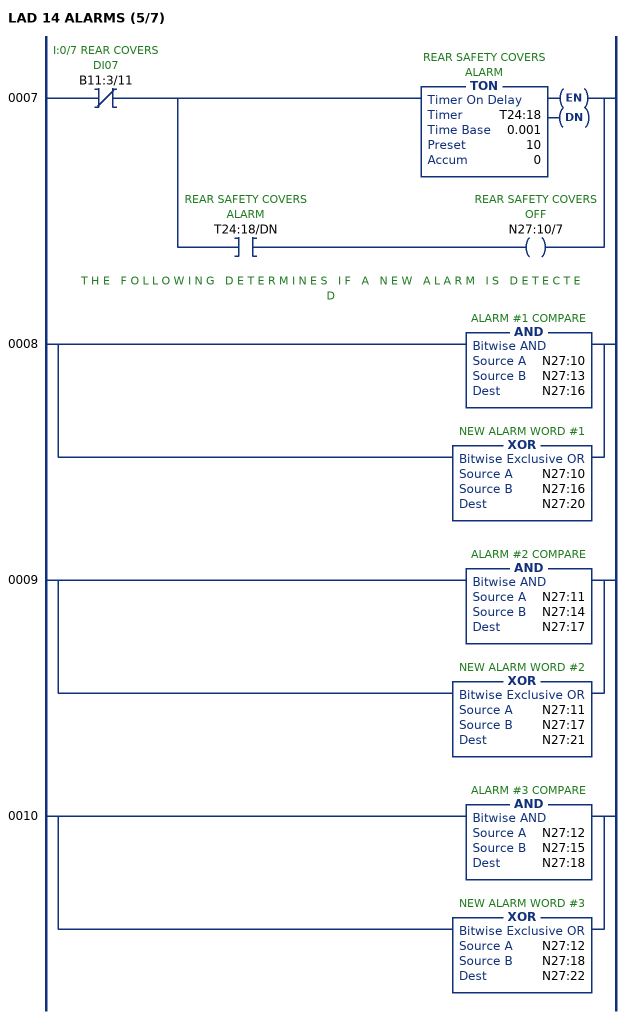
% Rung: 7 %
SOR XIO B11:3/11 BST TON T24:18 0.001 10 0 NXB XIC T24:18/DN OTE N27:10/7 BND EOR
%   B11:3/11  DI07  "I:0/7 REAR COVERS" %
%   T24:18  "REAR SAFETY COVERS ALARM" %
%   N27:10/7  "REAR SAFETY COVERS OFF" %
% Rung: 8 %
%        T H E   F O L L O W I N G   D E T E R M I N E S   I F   A   N E W   A L A R M   I S   D E T E C T E D %
SOR BST AND N27:10 N27:13 N27:16 NXB XOR N27:10 N27:16 N27:20 BND EOR
%   N27:10  "ALARM WORD #1 CURRENT" %
%   N27:13  "ALARM WORD #1 LAST SCAN" %
%   N27:16  "ALARM #1 COMPARE" %
%   N27:20  "NEW ALARM WORD #1" %
% Rung: 9 %
SOR BST AND N27:11 N27:14 N27:17 NXB XOR N27:11 N27:17 N27:21 BND EOR
%   N27:11  "ALARM WORD #2 CURRENT" %
%   N27:14  "ALARM WORD #2 LAST SCAN" %
%   N27:17  "ALARM #2 COMPARE" %
%   N27:21  "NEW ALARM WORD #2" %
% Rung: 10 %
SOR BST AND N27:12 N27:15 N27:18 NXB XOR N27:12 N27:18 N27:22 BND EOR
%   N27:12  "ALARM WORD #3 CURRENT" %
%   N27:15  "ALARM WORD #3 LAST SCAN" %
%   N27:18  "ALARM #3 COMPARE" %
%   N27:22  "NEW ALARM WORD #3" %

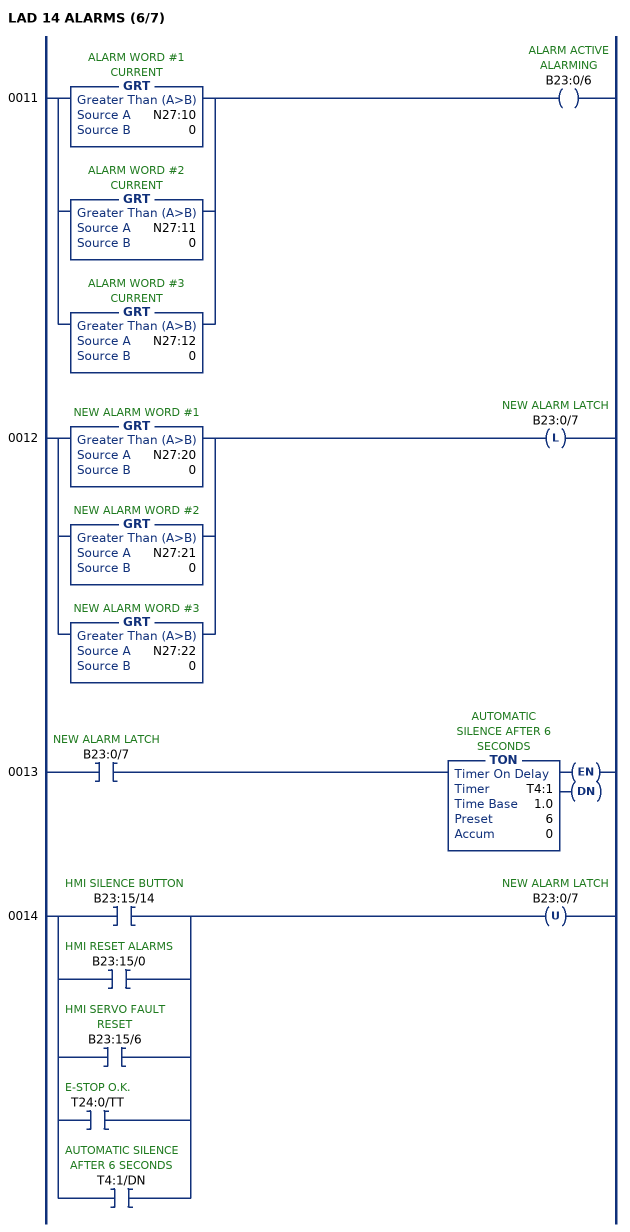
% Rung: 11 %
SOR BST GRT N27:10 0 NXB GRT N27:11 0 NXB GRT N27:12 0 BND OTE B23:0/6 EOR
%   N27:10  "ALARM WORD #1 CURRENT" %
%   N27:11  "ALARM WORD #2 CURRENT" %
%   N27:12  "ALARM WORD #3 CURRENT" %
%   B23:0/6  ALARMING  "ALARM ACTIVE" %
% Rung: 12 %
SOR BST GRT N27:20 0 NXB GRT N27:21 0 NXB GRT N27:22 0 BND OTL B23:0/7 EOR
%   N27:20  "NEW ALARM WORD #1" %
%   N27:21  "NEW ALARM WORD #2" %
%   N27:22  "NEW ALARM WORD #3" %
%   B23:0/7  "NEW ALARM LATCH" %
% Rung: 13 %
SOR XIC B23:0/7 TON T4:1 1.0 6 0 EOR
%   B23:0/7  "NEW ALARM LATCH" %
%   T4:1  "AUTOMATIC SILENCE AFTER 6 SECONDS" %
% Rung: 14 %
SOR BST XIC B23:15/14 NXB XIC B23:15/0 NXB XIC B23:15/6 NXB XIC T24:0/TT NXB XIC T4:1/DN BND OTU B23:0/7 EOR
%   B23:15/14  "HMI SILENCE BUTTON" %
%   B23:15/0  "HMI RESET ALARMS" %
%   B23:15/6  "HMI SERVO FAULT RESET" %
%   T24:0  "E-STOP O.K." %
%   T4:1  "AUTOMATIC SILENCE AFTER 6 SECONDS" %
%   B23:0/7  "NEW ALARM LATCH" %

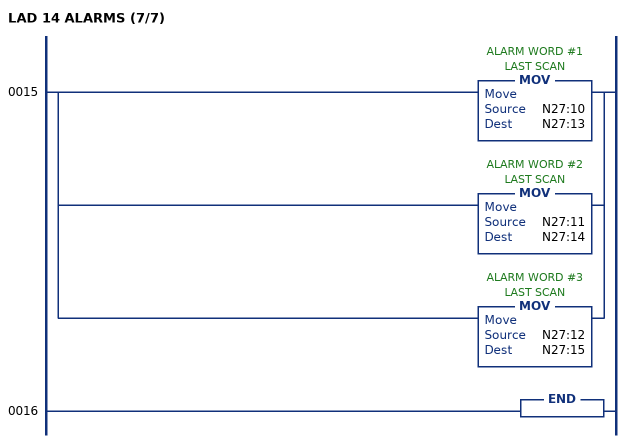
% Rung: 15 %
SOR BST MOV N27:10 N27:13 NXB MOV N27:11 N27:14 NXB MOV N27:12 N27:15 BND EOR
%   N27:10  "ALARM WORD #1 CURRENT" %
%   N27:13  "ALARM WORD #1 LAST SCAN" %
%   N27:11  "ALARM WORD #2 CURRENT" %
%   N27:14  "ALARM WORD #2 LAST SCAN" %
%   N27:12  "ALARM WORD #3 CURRENT" %
%   N27:15  "ALARM WORD #3 LAST SCAN" %
% Rung: 16 %
SOR END EOR

OTHER DOCUMENTED ADDRESSES
  B3:0/1  "ALL SUCTION COMPLETE SIDE 2"
  B3:0/3  "ALL DEPOSIT COMPLETE SIDE 2"
  B3:0/4  "ALL DEPOSIT COMPLETE BOTH SIDES"
  B3:0/7  "O/S"
  B3:0/8  "DEPOSIT COMPLETE SIDE 2 O/S"
  B3:0/14  "HMI HEATER #1 ON/OFF"
  B3:1/0  "O/S"
  B3:1/1  "deposit timing dn o/s"
  B3:1/2  "O/S"
  B3:1/3  "SUCTION TIME O/S"
  B11:0/3  "I:0/9 AIR PRESSURE"
  B11:0/4  "I:0/ NC/NF"
  B11:0/5  "I:0/ CONVEYOR FLIGHT DETECT"
  B11:0/7  "I:0/8 BRIDGE UP SENSOR"
  B11:0/8  "I:0/ CUSTOMER PERMISSIVE RUN ENERGIZE TO STOP DEPOSITOR"
  B11:0/9  "I:0/ LINER READY (CLEAR)"
  B11:0/10  "I:0/10 CYCLE START/STOP BUTTON"
  B11:0/14  "I:0/ OFF SWITCH"
  B11:1/1  "I:0/ DC POWER O.K."
  B11:1/2  "I:0/17 SERVO IN MOTION"
  B11:1/3  "I:0/ SERVO FAULT"
  B11:1/4  "I:0/ SERVO OUT 3"
  B11:1/5  "I:0/ SERVO OUT 4"
  B11:1/7  "I:0/ END OF TRAVEL SERVO FWD"
  B11:1/8  "I:0/ END OF TRAVEL SERVO REV"
  B11:1/9  "OILER OIL LOW SENSOR"
  B11:1/10  "OILER OIL HIGH SENSOR"
  B11:1/13  "I:0/ E-STOP #3"
  B11:1/14  "I:0/ E-STOP #4"
  B11:1/15  "I:0/ E-STOP #5"
  B11:2/1  "I:0/ E-STOP #7"
  B11:2/2  "I:0/ E-STOP #8"
  B11:2/3  "I:0/5 SAFETY SENSORS"
  B11:2/4  "I:0/6 SAFETY RIGHT COVER"
  B11:2/5  "I:0/7 TILT HOPPER"
  B11:2/7  "I:0/18 SAFETY DOORS"
  B11:2/8  "I:0/ SAFETY COVER #5"
  B12:0/0  "space holder"
  B12:0/3  "O:0/7 SPOUT OPEN"
  B12:0/4  "O:0/ SPOUT OPEN BANK #2"
  B12:0/5  "O:0/ SPOUT OPEN BANK #3"
  B12:0/6  "O:0/6 BLOWOFF"
  B12:0/7  "E-STOP SHUTOFF"
  B12:0/8  "MAPPIND DO GO SIGNAL"
  B12:0/10  "O:0/2 GREEN LIGHT"
  B12:0/11  DO12  "O:1/2 AMBER LIGHT"
  B12:0/13  "O:0/1 HORN"
  B12:0/14  DO18  "O:1/8 SERVO ENABLE"
  B12:0/15  "O:0/14 SERVO INDEX SIGNAL"
  B12:1/1  "O:0/ SERVO REGISTRATION SENSOR"
  B12:1/2  "O:0/ SERVO START HOMING"
  B12:1/3  "O:0/ SERVO HOME SWITCH"
  B12:1/4  "O:1/12 SERVO PRESET SELECT 0"
  B12:1/5  DO113  "O:1/13 SERVO PRESET SELECT 1"
  B12:1/6  "O:0/ SERVO PRESET SELECT 2"
  B12:1/7  "O:0/ SERVO PRESET SELECT 3"
  B12:1/8  "MAPPIND DO READY FOR PAN SIGNAL TO CUSTOMER"
  B12:1/11  "MAPPING DO BRIDGE UP"
  B12:1/12  "O:0/ CYCLE START LIGHT"
  B12:1/13  "O:0/8 BRIDGE DOWN"
  B12:1/14  "MAPPING OILER"
  B12:1/15  "MAPPING DO LINER PLACER GO SIGNAL"
  B12:2/1  "MAPPING DO VFD #1 START"
  B12:2/2  "MAPPING DO VFD #2 ENABLE"
  B12:2/3  "MAPPING DO VFD #2 START"
  B12:2/4  "MAPPING DO VFD #3 ENABLE"
  B12:2/5  "MAPPING DO VFD #3 START"
  B13:0/4  "FORCE OUTPUT O:0/4"
  B13:0/6  "FORCE OUTPUT O:0/6"
  B13:0/7  "FORCE OUTPUT O:0/7"
  B13:0/8  "FORCE OUTPUT O:0/8"
  B13:0/9  "FORCE OUTPUT O:0/9"
  B13:0/10  "FORCE OUTPUT O:0/10"
  B13:0/11  "FORCE OUTPUT O:0/11"
  B13:0/12  "FORCE OUTPUT O:0/12"
  B13:0/13  "FORCE OUTPUT O:0/13"
  B13:0/14  "FORCE OUTPUT O:0/14"
  B13:0/15  "FORCE OUTPUT O:0/15"
  B13:1/0  "FORCE OUTPUT O:1/0"
  B13:1/1  "FORCE OUTPUT O:1/1"
  B13:1/2  "FORCE OUTPUT O:1/2"
  B13:1/3  "FORCE OUTPUT O:1/3"
  B13:1/4  "FORCE OUTPUT O:1/4"
  B13:1/5  "FORCE OUTPUT O:1/5"
  B13:1/6  "FORCE OUTPUT O:1/6"
  B13:1/7  "FORCE OUTPUT O:1/7"
  B13:1/8  "FORCE OUTPUT O:1/8"
  B13:1/9  "FORCE OUTPUT O:1/9"
  B13:1/10  "FORCE OUTPUT O:1/10"
  B13:1/11  "FORCE OUTPUT O:1/11"
  B13:1/12  "FORCE OUTPUT O:1/12"
  B13:1/13  "FORCE OUTPUT O:1/13"
  B13:1/14  "FORCE OUTPUT O:1/14"
  B13:1/15  "FORCE OUTPUT O:1/15"
  B13:2/10  "FORCE OUTPUT O:2/10"
  B13:2/11  "FORCE OUTPUT O:2/11"
  B13:2/12  "FORCE OUTPUT O:2/12"
  B13:2/13  "FORCE OUTPUT O:2/13"
  B13:2/14  "FORCE OUTPUT O:2/14"
  B13:2/15  "FORCE OUTPUT O:2/15"
  B13:3/0  "FORCE OUTPUT O:3/0"
  B13:3/1  "FORCE OUTPUT O:3/1"
  B13:3/2  "FORCE OUTPUT O:3/2"
  B13:3/3  "FORCE OUTPUT O:3/3"
  B13:3/4  "FORCE OUTPUT O:3/4"
  B13:3/5  "FORCE OUTPUT O:3/5"
  B13:3/6  "FORCE OUTPUT O:3/6"
  B13:3/7  "FORCE OUTPUT O:3/7"
  B13:3/8  "FORCE OUTPUT O:3/8"
  B13:3/9  "FORCE OUTPUT O:3/9"
  B13:3/10  "FORCE OUTPUT O:3/10"
  B13:3/11  "FORCE OUTPUT O:3/11"
  B13:3/12  "FORCE OUTPUT O:3/12"
  B13:3/13  "FORCE OUTPUT O:3/13"
  B13:3/14  "FORCE OUTPUT O:3/14"
  B13:3/15  "FORCE OUTPUT O:3/15"
  B13:4/0  "FORCE OUTPUT O:4/0"
  B13:4/1  "FORCE OUTPUT O:4/1"
  B13:4/2  "FORCE OUTPUT O:4/2"
  B13:4/3  "FORCE OUTPUT O:4/3"
  B13:4/4  "FORCE OUTPUT O:4/4"
  B13:4/5  "FORCE OUTPUT O:4/5"
  B13:4/6  "FORCE OUTPUT O:4/6"
  B13:4/7  "FORCE OUTPUT O:4/7"
  B13:4/8  "FORCE OUTPUT O:4/8"
  B13:4/9  "FORCE OUTPUT O:4/9"
  B13:4/10  "FORCE OUTPUT O:4/10"
  B13:4/11  "FORCE OUTPUT O:4/11"
  B13:4/12  "FORCE OUTPUT O:4/12"
  B13:4/13  "FORCE OUTPUT O:4/13"
  B13:4/14  "FORCE OUTPUT O:4/14"
  B13:4/15  "FORCE OUTPUT O:4/15"
  B13:5/0  "FORCE OUTPUT O:5/0"
  B13:5/1  "FORCE OUTPUT O:5/1"
  B13:5/2  "FORCE OUTPUT O:5/2"
  B13:5/3  "FORCE OUTPUT O:5/3"
  B13:5/4  "FORCE OUTPUT O:5/4"
  B13:5/5  "FORCE OUTPUT O:5/5"
  B13:5/6  "FORCE OUTPUT O:5/6"
  B13:5/7  "FORCE OUTPUT O:5/7"
  B13:5/8  "FORCE OUTPUT O:5/8"
  B13:5/9  "FORCE OUTPUT O:5/9"
  B13:5/10  "FORCE OUTPUT O:5/10"
  B13:5/11  "FORCE OUTPUT O:5/11"
  B13:5/12  "FORCE OUTPUT O:5/12"
  B13:5/13  "FORCE OUTPUT O:5/13"
  B13:5/14  "FORCE OUTPUT O:5/14"
  B13:5/15  "FORCE OUTPUT O:5/15"
  B15:2/0  "AGITATOR ENABLED"
  B23:0/1  "DEPOSIT TRIGGER POSITION #1 O/S"
  B23:0/8  "O/S"
  B23:0/9  "O/S"
  B23:0/12  "RECIPE CHANGED O/S"
  B23:1/2  "STATUS SUBROUTINE"
  B23:1/3  "O/S"
  B23:1/4  "CYCLE START/STOP BUTTON O/S"
  B23:1/5  "CYCLE STOP PUSHBUTTON"
  B23:1/8  "CYCLE STARTING"
  B23:1/10  "CYCLE STOPPING"
  B23:1/11  "CYCLE STOPPED"
  B23:1/12  "MAIN CYL SUCTION"
  B23:1/13  B  "DEC2HEX FL SUBROUTINE"
  B23:1/14  "DEC2HEX SD SUBROUTINE"
  B23:1/15  "CONFIRMATION PASS CHANGED"
  B23:2/0  "CHANGE PSWRD YES/NO VISIBILITY"
  B23:2/1  "CHANGE PASSWORD ? YES !"
  B23:2/2  "CHANGE PASSWORD ? NO !"
  B23:2/3  "HMI LOGOUT BUTTON"
  B23:2/4  "NEW PASSWORD VISIBILITY BIT"
  B23:2/5  "VFD'S SUBROUTINE"
  B23:2/8  "RECIPE SELECT SUBROUTINE"
  B23:2/9  "NC/NF SUBROUTINE"
  B23:2/10  "FLIGHT DETECT O/S"
  B23:2/11  "O/S"
  B23:2/12  "PAN DETECTED"
  B23:2/13  "SERVO SUBROUTINE"
  B23:2/14  "O/S"
  B23:2/15  "VFD ANALOG SPEED REF SUBROUTINE"
  B23:3/0  "MAPPING ANALOG INPUTS SUBROUTINE"
  B23:3/1  "SERVO JOGGING"
  B23:3/2  "O/S"
  B23:3/3  "SERVO MOVING O/S"
  B23:3/4  "O/S"
  B23:3/5  "SERVO STOPPED O/S"
  B23:3/6  "EVERYTHING GO LATCH"
  B23:3/9  "SEQUENCER SUBROUTINE"
  B23:3/11  "O/S"
  B23:3/12  "MAPPING ANALOG OUTPUTS SUBROUTINE"
  B23:3/14  "DONE SIGNAL"
  B23:3/15  "O/S"
  B23:4/0  "CYCLE TIME DONE O/S"
  B23:4/2  "SERVO INDEX LATCH"
  B23:4/5  "LOGIN SUBROUTINE"
  B23:4/6  "LINER SUBROUTINE"
  B23:4/7  "ALWAYS OPEN REMOVE FOR PANELVIEW PLUS"
  B23:4/8  "OILER SUBROUTINE"
  B23:4/9  "O/S"
  B23:4/10  "TRIGGER OILER O/S"
  B23:4/11  "O/S"
  B23:4/12  "OIL LATCH"
  B23:4/13  "SERVO ACTUATOR SUBROUTINE"
  B23:4/14  "CHANGE PASSWORD VISIBILITY"
  B23:4/15  "CHANGE PASSWORD YES"
  B23:5/0  "RESET PASSWORDS"
  B23:5/1  "C-MORE HMI BEEP"
  B23:5/3  "C-MORE HMI NO ACCESS POPUP WINDOW"
  B23:5/4  "NO ACCESS SCENERIO 1"
  B23:5/5  "NO ACCESS SCENERIO 2"
  B23:5/6  "NO ACCESS SCENERIO 3"
  B23:5/7  "NO ACCESS SCENERIO 4"
  B23:5/8  "NO ACCESS SCENERIO 5"
  B23:5/9  "NO ACCESS SCENERIO 6"
  B23:5/10  "NO ACCESS SCENERIO 7"
  B23:5/11  "NO ACCESS SCENERIO 8"
  B23:5/12  "LATCH PAUSE MODE"
  B23:6/2  "O/S"
  B23:6/3  "O/S"
  B23:6/5  "DEPOSITOR SEQUENCER STEP #1"
  B23:6/6  "DEPOSITOR SEQUENCER STEP #2"
  B23:6/7  "DEPOSITOR SEQUENCER STEP #3"
  B23:6/8  "DEPOSITOR SEQUENCER STEP #4"
  B23:6/9  "DEPOSITOR SEQUENCER STEP #5"
  B23:6/10  "DEPOSITOR SEQUENCER STEP #6"
  B23:6/11  "DEPOSITOR SEQUENCER STEP #7"
  B23:6/12  "DEPOSITOR SEQUENCER STEP #8"
  B23:6/13  "DEPOSITOR SEQUENCER STEP #9"
  B23:6/14  "DEPOSITOR SEQUENCER STEP #10"
  B23:6/15  "DEPOSITOR SEQUENCER STEP #11"
  B23:7/0  "DEPOSITOR SEQUENCER STEP #12"
  B23:7/1  "DEPOSITOR SEQUENCER STEP #13"
  B23:7/2  "DEPOSITOR SEQUENCER STEP #14"
  B23:7/3  "DEPOSITOR SEQUENCER STEP #15"
  B23:7/4  "DEPOSITOR SEQUENCER STEP #16"
  B23:7/5  "DEPOSITOR SEQUENCER STEP #17"
  B23:7/6  "DEPOSITOR SEQUENCER STEP #18"
  B23:7/7  "DEPOSITOR SEQUENCER STEP #19"
  B23:7/8  "DEPOSITOR SEQUENCER STEP #20"
  B23:10  "1ST WORD BIT SHIFT"
  B23:11  "2ND WORD BIT SHIFT"
  B23:12  "3RD WORD BIT SHIFT"
  B23:15  "HMI BITS"
  B23:15/1  "HMI PRIME SELECT"
  B23:15/2  "HMI OFF SELECT"
  B23:15/3  "HMI AUTO SELECT"
  B23:15/4  "HMI CYCLE START"
  B23:15/5  "HMI CYCLE STOP"
  B23:15/7  "HMI SERVO JOG FWD"
  B23:15/8  "HMI SERVO JOG REV"
  B23:15/9  "HMI CLEAN MODE"
  B23:15/10  "HMI DEPOSITOR ON/OFF"
  B23:15/11  "HMI WIPE SCREEN"
  B23:15/12  "NC/NF ALWAYS ON"
  B23:15/13  "HMI DOUBLE CYCLE DEPOSITOR ON/OFF"
  B23:15/15  "IGNORE CUSTOMER PERMISSIVE RUN SIGNAL"
  B23:16  "HMI BITS"
  B23:16/0  "HMI FORCE DEPOSIT TRIGGER"
  B23:16/4  "HMI LINER PLACER ON/OFF"
  B23:16/5  "HMI SPEED OF MACHINE CALC ON/OFF"
  B23:16/7  "HMI BRIDGE DOWN FORCE"
  B23:16/8  "HMI BRIDGE ON/OFF"
  B23:16/9  "HMI OILER ON/OFF"
  B23:16/12  "HMI VFD #1 ON/OFF"
  B23:16/13  "HMI FORCE VFD #1"
  B23:16/14  "HMI VFD #2 ON/OFF"
  B23:16/15  "HMI FORCE VFD #2"
  B23:17  "HMI BITS"
  B23:17/0  "HMI VFD #3 ON/OFF"
  B23:17/1  "HMI FORCE VFD #3"
  B23:17/2  "HMI START HOMING SERVO"
  B23:17/3  "HMI RESET TOTAL PAN COUNT"
  B23:17/4  "SET DATE & TIME"
  B23:17/5  "HMI DEFINE HOME"
  B50:0  "DIGITAL INPUT STATUS"
  B50:2  "START HOMING"
  B50:3  "DEFINE HOME"
  B50:4  "RESET DRIVE"
  C5:0  "ROW COUNTER"
  C5:1  "deposit time indexer"
  C5:3  "DEPOSIT COUNT"
  C25:0  "CPM COUNTER"
  C25:1  "DEPOSIT COUNT"
  C25:2  "SERVO INDEX COUNTER"
  C25:3  "TRANSFER PARAMETER TIMER"
  C25:4  "OIL SPRAY COUNTER"
  C25:5  "SERVO MESSAGE STATEMENT COUNTER"
  D0206  
  DFILE:0  "OUTPUT"
  DFILE:1  "INPUT"
  DFILE:2  "STATUS"
  DFILE:3  "BINARY"
  DFILE:4  "TIMER"
  DFILE:5  "COUNTER"
  DFILE:6  "CONTROL"
  DFILE:7  "INTEGER"
  DFILE:8  "FLOAT"
  DFILE:9  "HEATER"
  DFILE:10  "MAP AO"
  DFILE:11  "MAP DI"
  DFILE:12  "MAP DO"
  DFILE:13  "FORCE OUT"
  DFILE:20  "VFD'S"
  DFILE:21  "VFD'S"
  DFILE:23  "TYPICAL"
  DFILE:24  "TYPICAL"
  DFILE:25  "TYPICAL"
  DFILE:26  "VFD'S"
  DFILE:27  "TYPICAL"
  DFILE:28  "TYPICAL"
  F8:0  "CUSTOMER SPEED REFERENCE"
  F8:1  "MULTIPLIER"
  F8:2  "ROWS PER PAN"
  F8:3  "PAN 1 2 OZ PAN SUCTION DELAY"
  F8:4  "PAN 2 4 OZ PAN SUCTION DELAY"
  F8:5  "PAN 3 MINI PAN SUCTION DELAY"
  F28:0  "Multiplier for 1" move Index 0 Distance"
  F28:1  "Multiplier 1 ft per sec Index 0 Velocity"
  F28:2  "AVERAGE CURRENT"
  F28:4  "Multiplier Acc/Dec Same as F28:0"
  F28:5  "STORAGE HOLD FOR 1ST ROW"
  F28:6  "FIRST ROW DISTANCE ADDER"
  F28:10  "HMI ACCELERATION MULTIPLIER INDEX 0"
  F28:11  "HMI DECELERATION MULTIPLIER INDEX 0"
  F28:12  "HMI ACCELERATION MULTIPLIER INDEX 1"
  F28:13  "HMI DECELERATION MULTIPLIER INDEX 1"
  F28:16  "CONSTANT CALIBRATED VARIABLE"
  F28:20  "TOTAL PAN COUNT"
  F28:21  "PPM CURRENT"
  F28:22  "PPM PREVIOUS"
  F28:23  "CPM CURRENT"
  F28:24  "CPM PREVIOUS"
  F28:30  "CMORE RECIPE MODIFYING TEMP FILES"
  F98:0  "CURRENT RECIPE 1ST ROW DISTANCE"
  F98:1  "CURRENT RECIPE VELOCITY 1ST ROW"
  F98:2  "CURRENT RECIPE DISTANCE ROW TO ROW"
  F98:3  "CURRENT RECIPE VELOCITY ROW TO ROW"
  F98:4  "MOTION DELAY"
  F101:6  "DECIMAL PASSED # TO CONVERT TO HEX"
  I:2.0  "THERMOCOUPLE #1"
  L52:0  "INDEX O DISTANCE"
  L52:1  "INDEX 0 VELOCITY"
  L52:2  "INDEX 0 ACCEL"
  L52:3  "INDEX 0 DECEL"
  L52:4  "INDEX 1 DISTANCE"
  L52:5  "INDEX 1 VELOCITY"
  L52:6  "INDEX 1 ACCEL"
  L52:7  "INDEX 1 DECEL"
  L52:8  "SERVO DRIVE FAULT STATUS L20:108"
  L52:9  "MESSAGE ON/OFF"
  L52:12  "SPEED SETTING FROM HMI CONVERTED TO DRIVE UNITS"
  L52:20  "VALUE CHANGED"
  L52:21  "VALUE CHANGED"
  L52:22  "VALUE CHANGED"
  L52:23  "VALUE CHANGED"
  L52:24  "VALUE CHANGED"
  L52:25  "VALUE CHANGED"
  L52:26  "VALUE CHANGED"
  L52:27  "VALUE CHANGED"
  MG53:0  "INDEX 0 REGISTRATION DISTANCE"
  MG53:1  "INDEX 0 VELOCITY"
  MG53:2  "INDEX 0 ACCEL"
  MG53:3  "INDEX 0 DECEL"
  MG53:4  "INDEX 1 DISTANCE"
  MG53:5  "INDEX 1 VELOCITY"
  MG53:6  "INDEX 1 ACCEL"
  MG53:7  "INDEX 1 DECEL"
  MG53:8  "FAULT STATUS"
  MG53:9  "RESET DRIVE"
  MG53:10  "START HOMING"
  MG53:11  "DEFINE HOME"
  MG53:12  "CURRENT LIMIT FORWARD"
  MG53:13  "CURRENT LIMIT REVERSE"
  MG53:14  "HOST CONTROL MODE"
  MG53:15  "HOST INDEX"
  MG53:16  "AVERAGE CURRENT"
  MG53:17  "DIGITAL INPUT STATUS"
  MG53:18  "OPERATION MODE"
  MG53:20  "MOTOR POSITION IN COUNTS"
  MG70:0  "INITIAL TIMEOUT SETUP FOR VFD #1"
  MG70:1  "WRITE VFD #1 COMMANDS 3 WORDS"
  MG70:2  "READ VFD #1 STATUS 3 WORDS"
  MG70:3  "INITIAL TIMEOUT SETUP FOR VFD #2"
  MG70:4  "WRITE VFD #2 COMMANDS 3 WORDS"
  MG70:5  "READ VFD #2 STATUS 3 WORDS"
  MG70:6  "INITIAL TIMEOUT SETUP FOR VFD #3"
  MG70:7  "WRITE VFD #3 COMMANDS 3 WORDS"
  MG70:8  "READ VFD #3 STATUS 3 WORDS"
  N7:0  "HMI BRIDGE ENABLE"
  N7:0/0  "0"
  N7:0/1  "1"
  N7:0/2  "2"
  N7:1  "FIFO #0"
  N7:11  "# OF ROWS"
  N27:1  "RECIPE SELECTED"
  N27:2  "INDIRECT ADDRESSING RECIPE SELECTED"
  N27:3  "PREVIOUS RECIPE SELECTED"
  N27:4  "BINARY CONTROL OF SERVO INDEXES"
  N27:5  "HMI DISPLAY MACHINE STATUS"
  N27:6  "HMI SUCTION DELAY TIMER"
  N27:7  "HMI DEPOSIT DELAY TIMER"
  N27:8  "CURRENT SCREEN"
  N27:9  "FORCED SCREEN"
  N27:10/0  "ALARM #0"
  N27:10/8  "SUCTION #2 PNEUMATIC FAILURE"
  N27:10/9  "ALARM #9"
  N27:10/10  "ALARM #10"
  N27:10/11  "E-STOP PRESSED MAIN ENCL"
  N27:10/12  "E-STOP PRESSED MAIN ENCL"
  N27:10/13  "SAFETY DOOR NEAR"
  N27:10/14  "TILT HOPPER"
  N27:10/15  "HOPPER COVER"
  N27:11/0  "ALARM #16"
  N27:11/1  "ALARM #17"
  N27:11/2  "ALARM #18"
  N27:11/3  "ALARM #19"
  N27:11/4  "VFD #2 FAULT ALARM"
  N27:11/5  "VFD #3 FAULT ALARM"
  N27:19  "ENSURE ZERO NOT PUT IN DIV STATEMENT"
  N27:24  "HMI # OF OIL SPRAYS"
  N27:25  "NEW PERSON LOGGED IN"
  N27:30  "RECIPE SELECTED FOR MODIFYING"
  N27:31  "INDIRECT RECIPE FOR MODIFYING"
  N27:40  "User 1=ADMIN, 2=MAINT, 3=LEAD, 4=OPER, 5=TEMP 88=BACKDOOR 99=HBTECH"
  N27:41  "ADMIN PASSWORD"
  N27:42  "MAINT PASSWORD"
  N27:43  "LEAD PASSWORD"
  N27:44  "OPER PASSWORD"
  N27:45  "TEMP PASSWORD"
  N27:46  "ADMIN BACKDOOR"
  N27:48  "BACKDOOR PASSWORD"
  N27:49  "HB TECH PASSWORD"
  N27:50  "NEW PASSWORD TEMPORARY STORAGE"
  N27:52  "OLD PASSWORD TEMPORARY STORAGE"
  N27:53  "PASSWORD ENTERED BY CLIENT"
  N27:54  "PERSON LOGGED IN"
  N27:60  "PLC YEAR"
  N27:61  "PLC MONTH"
  N27:62  "PLC DAY"
  N27:63  "PLC HOUR"
  N27:64  "PLC MINUTE"
  N27:65  "PLC SECOND"
  N27:70  "SET YEAR"
  N27:71  "SET MONTH"
  N27:72  "SET DAY"
  N27:73  "SET HOUR"
  N27:74  "SET MINUTE"
  N27:75  "SET SECONDS"
  N27:100  "ACCESS CONTROL SCREEN #"
  N27:101  "GRANT ACCESS TO THIS PERSON"
  N27:102  "GRANT ACCESS TO THIS PERSON"
  N27:103  "GRANT ACCESS TO THIS PERSON"
  N27:104  "GRANT ACCESS TO THIS PERSON"
  N27:105  "GRANT ACCESS TO THIS PERSON"
  N27:110  "ACCESS CONTROL SCREEN #"
  N27:111  "GRANT ACCESS TO THIS PERSON"
  N27:112  "GRANT ACCESS TO THIS PERSON"
  N27:113  "GRANT ACCESS TO THIS PERSON"
  N27:114  "GRANT ACCESS TO THIS PERSON"
  N27:115  "GRANT ACCESS TO THIS PERSON"
  N27:120  "ACCESS CONTROL SCREEN #"
  N27:121  "GRANT ACCESS TO THIS PERSON"
  N27:122  "GRANT ACCESS TO THIS PERSON"
  N27:123  "GRANT ACCESS TO THIS PERSON"
  N27:124  "GRANT ACCESS TO THIS PERSON"
  N27:125  "GRANT ACCESS TO THIS PERSON"
  N27:130  "ACCESS CONTROL SCREEN #"
  N27:131  "GRANT ACCESS TO THIS PERSON"
  N27:132  "GRANT ACCESS TO THIS PERSON"
  N27:133  "GRANT ACCESS TO THIS PERSON"
  N27:134  "GRANT ACCESS TO THIS PERSON"
  N27:135  "GRANT ACCESS TO THIS PERSON"
  N27:140  "ACCESS CONTROL SCREEN #"
  N27:141  "GRANT ACCESS TO THIS PERSON"
  N27:142  "GRANT ACCESS TO THIS PERSON"
  N27:143  "GRANT ACCESS TO THIS PERSON"
  N27:144  "GRANT ACCESS TO THIS PERSON"
  N27:145  "GRANT ACCESS TO THIS PERSON"
  N27:150  "ACCESS CONTROL SCREEN #"
  N27:151  "GRANT ACCESS TO THIS PERSON"
  N27:152  "GRANT ACCESS TO THIS PERSON"
  N27:153  "GRANT ACCESS TO THIS PERSON"
  N27:154  "GRANT ACCESS TO THIS PERSON"
  N27:155  "GRANT ACCESS TO THIS PERSON"
  N27:160  "ACCESS CONTROL SCREEN #"
  N27:161  "GRANT ACCESS TO THIS PERSON"
  N27:162  "GRANT ACCESS TO THIS PERSON"
  N27:163  "GRANT ACCESS TO THIS PERSON"
  N27:164  "GRANT ACCESS TO THIS PERSON"
  N27:165  "GRANT ACCESS TO THIS PERSON"
  N27:170  "ACCESS CONTROL SCREEN #"
  N27:171  "GRANT ACCESS TO THIS PERSON"
  N27:172  "GRANT ACCESS TO THIS PERSON"
  N27:173  "GRANT ACCESS TO THIS PERSON"
  N27:174  "GRANT ACCESS TO THIS PERSON"
  N27:175  "GRANT ACCESS TO THIS PERSON"
  N37:11  "HOT OIL HIGH LIMIT"
  N37:12  "HOT OIL LOW LIMIT"
  N37:15  "HOT OIL ACTUAL TEMP"
  N37:16  "HEATER CONTROL BASED ON 10S TIME BASE"
  N47:4  "WRITE INITIALE VFD SETTINGS"
  N47:10  "READ VFD STATUS & SPEED REF"
  N51:0  "INDEX # TO BE PERFORMED"
  N51:1  "OPERATION MODE 2 = PRESET VEL 7 = INDEXING"
  N51:3  "CURRENT LIMIT FORWARD"
  N51:4  "CURRENT LIMIT REVERSE"
  N51:5  "DRIVE SPEED IN % OF MAX"
  N51:6  "BELT SPEED ACTUAL TO HMI DISPLAY"
  N51:10  "VALUE CHANGED"
  N51:13  "VALUE CHANGED"
  N51:14  "VALUE CHANGED"
  N77:3  "INITIAL STATE FOR VFD'S"
  N77:10  "LOGIC WORD COMMAND TO VFD#1"
  N77:10/0  "STOP VFD #1"
  N77:10/1  "START VFD #1"
  N77:10/3  "RESET VFD #1 FAULT"
  N77:12  "SPEED CMD SENT TO VFD #1"
  N77:13  "HMI SPEED CMD FOR VFD#1"
  N77:14  "STATUS WORD FROM VFD#1"
  N77:14/6  "ALARM BIT FROM VFD #1"
  N77:14/7  "FAULT BIT FROM VFD #1"
  N77:16  "SPEED FEEDBACK SENT FROM VFD#1"
  N77:17  "HMI SPEED FEEDBACK VFD #1"
  N77:20  "LOGIC WORD COMMAND TO VFD#2"
  N77:20/0  "STOP VFD #2"
  N77:20/1  "START VFD #2"
  N77:20/3  "RESET VFD #1 FAULT"
  N77:22  "SPEED CMD SENT TO VFD #2"
  N77:23  "HMI SPEED CMD FOR VFD#2"
  N77:24  "STATUS WORD FROM VFD#2"
  N77:24/6  "ALARM BIT FROM VFD #2"
  N77:24/7  "FAULT BIT FROM VFD #2"
  N77:26  "SPEED FEEDBACK SENT FROM VFD#2"
  N77:27  "HMI SPEED FEEDBACK VFD #2"
  N77:30  "LOGIC WORD COMMAND TO VFD#3"
  N77:30/0  "STOP VFD #3"
  N77:30/1  "START VFD #3"
  N77:30/3  "RESET VFD #1 FAULT"
  N77:32  "SPEED CMD SENT TO VFD #3"
  N77:33  "HMI SPEED CMD FOR VFD#3"
  N77:34  "STATUS WORD FROM VFD#3"
  N77:34/6  "ALARM BIT FROM VFD #3"
  N77:34/7  "FAULT BIT FROM VFD #3"
  N77:36  "SPEED FEEDBACK SENT FROM VFD#3"
  N77:37  "HMI SPEED FEEDBACK VFD #3"
  N100:0  "PASSED CHECKSUM VALUE FOR HOST COMMAND PREFIX"
  PD9:1  "HOT OIL HEATER"
  R6:0  "ASCII WRITE INSTRUCTION"
  R6:0/DN  "ASCII Write instruction complete"
  R6:1  "NC/NF BIT SHIFT REGISTER"
  R6:2  "FIFO DEPOSITING TIME"
  R6:3  "SUCTION FIFO CONTROL WORD"
  ST99:29  "RECIPE NAME MODIFY"
  ST102:0  "PASSED HOST COMMAND STRING PREFIX"
  ST102:1  "0' (USED IF VARIABLE IS LESS THEN CURRENT HEX PLACE)"
  ST102:2  "DEC2HEX SUBROUTINE OUTPUT"
  ST102:3  "XFFFF DEC2HEX CONV"
  ST102:4  "XXFFF DEC2HEX CONV"
  ST102:5  "XXXFF DEC2HEX CONV"
  ST102:6  "XXXXF DEC2HEX CONV"
  ST102:7  "XXXXX DEC2HEX CONV"
  ST102:8  "A'"
  ST102:9  "B'"
  ST102:10  "C'"
  ST102:11  "D'"
  ST102:12  "E'"
  ST102:13  "F'"
  ST102:14  "HOST COMMAND STRING PREFIX + VARIABLE IN HEX"
  ST102:15  "STRING + 1 CHECKSUM VALUE"
  ST102:16  "STRING + 2 CHECKSUM VALUES (MINUS CARRIAGE RETURN)"
  ST102:17  "CARRIAGE RETURN"
  ST102:18  "COMPLETE STRING"
  ST104:0  "INDEX 0 DISTANCE"
  ST104:1  "INDEX 0 REGISTRATION"
  ST104:2  "INDEX 0 VELOCITY"
  ST104:3  "INDEX 0 ACCELERATION"
  ST104:4  "INDEX 0 DECELERATION"
  ST104:5  "INDEX 1 DISTANCE"
  ST104:6  "INDEX 1 REGISTRATION"
  ST104:7  "INDEX 1 VELOCITY"
  ST104:8  "INDEX 1 ACCELERATION"
  ST104:9  "INDEX 1 DECELERATION"
  T4:0  "TIME FOR CYLINDERS TO MOVE"
  T4:2  "DEPOSIT TRIGGER"
  T4:3  "TIME FOR CYLINDERS TO MOVE"
  T4:4  "SHIFT DELAY DEPOSIT #2"
  T4:5  "SHIFT DELAY SUCTION #2"
  T4:21  "HOT OIL HEATER ON BASED ON 10S TIMER"
  T24:2  "AUTO START VFD"
  T24:3  "SHIFT DELAY DEPOSIT #1"
  T24:4  "SHIFT DELAY SUCTION #1"
  T24:10  "CPM TIMER"
  T24:11  "E-STOP ALARM"
  T24:19  "SUCTION #2 PNEUMATIC FAILURE"
  T24:20  "DC POWER SUPPLY ALARM"
  T24:21  "PLC FAULTED"
  T24:22  "E-STOP PRESSED MAIN ENCL"
  T24:23  "E-STOP PRESSED MAIN ENCL"
  T24:24  "SAFETY DOOR NEAR"
  T24:25  "TILT HOPPER"
  T24:26  "HOPPER COVER"
  T24:27  "ALARM #16"
  T24:28  "ALARM #17"
  T24:29  "ALARM #18"
  T24:39  "STOP JOGGING BY DISABLING DRIVE BRIEFLY"
  T24:48  "WIPE SCREEN TIMER"
  T24:49  "VFD #1 ALARM/FAULT TIMER"
  T24:50  "VFD #2 ALARM/FAULT TIMER"
  T24:51  "VFD #3 ALARM/FAULT TIMER"
  T24:52  "OILER TRIGGER ON TIME"
  T24:53  "REPEAT OIL SPRAYS"
  T24:54  "SERVO HOMING TIMER"
  T24:55  "RESET PASSWORDS TIME DELAY"
  T24:56  "MACHINE SPEED CONTROL"
  T24:57  "E-STOP PRESSED SERVO DISCHARGING"
  T24:58  "SERVO DRIVE RESETTING DELAY"
  T24:60  "INITIATE SERVO MESSAGES"
  T24:61  "SEQUENCER TIME DELAY STEP #1"
  T24:62  "SEQUENCER TIME DELAY STEP #2"
  T24:63  "SEQUENCER TIME DELAY STEP #3"
  T24:64  "SEQUENCER TIME DELAY STEP #4"
  T24:65  "SEQUENCER TIME DELAY STEP #5"
  T24:66  "SEQUENCER TIME DELAY STEP #6"
  T24:66/DN  "SEQUENCER TIME DELAY STEP #6"
  T24:67  "SEQUENCER TIME DELAY STEP #7"
  T24:67/DN  "SEQUENCER TIME DELAY STEP #7"
  T24:68  "SEQUENCER TIME DELAY STEP #8"
  T24:69  "SEQUENCER TIME DELAY STEP #9"
  T24:70  "SEQUENCER TIME DELAY STEP #10"
  T24:71  "SEQUENCER TIME DELAY STEP #11"
  T24:72  "SEQUENCER TIME DELAY STEP #12"
  T24:73  "SEQUENCER TIME DELAY STEP #13"
  T24:74  "SEQUENCER TIME DELAY STEP #14"
  T24:75  "SEQUENCER TIME DELAY STEP #15"
  T24:76  "SEQUENCER TIME DELAY STEP #16"
  T24:77  "SEQUENCER TIME DELAY STEP #17"
  T24:78  "SEQUENCER TIME DELAY STEP #18"
  T24:79  "SEQUENCER TIME DELAY STEP #19"
  T24:80  "SEQUENCER TIME DELAY STEP #20"
  T24:82  "BLOWOFF TIMER"
  U:3  "DEPOSITOR SUBROUTINE"
  U:4  "SERVO SUBROUTINE"
  U:5  "RECIPE SELECT SUBROUTINE"
  U:6  "NC/NF SUBROUTINE"
  U:7  "VFD'S SUBROUTINE"
  U:8  "VFD ANALGO SPEED REFERENCE SUBROUTINE"
  U:10  "MAP SEQUENCER SUBROUTINE"
  U:13  "STATUS SUBROUTINE"
  U:15  "LOGIN SUBROUTINE"
  U:16  "OILER SUBROUTINE"
  U:17  "LINER SUBROUTINE"
  U:20  "SERVO ACTUATOR SUBROUTINE"
  U:31  "DEC2HEX FL SUBROUTINE"
  U:32  "DEC2HEX SD SUBROUTINE"
  XIC  

COMMENTS NOT ATTACHED TO A CURRENT RUNG
  N77:17: VFD #1 COMMANDS AND FEEDBACK
  N27:75: AS LONG AS THE CHANGE DATE AND TIME SCREEN IS NOT CURRENTLY OPEN THEN THE PLC WILL POPULATE THE TEMPORARY HOLD INTEGERS WITH THE CURRENT DATE AND TIME VALUES
  N27:65: T I M E    A N D    D A T E    H A N D S H A K I N G    F O R    O P E R A T O R    I N T E R F A C E
  N27:17: V F D    # 3
  MG40:2: This last Message reads the Drives Logic status and the speed Feedback and displays it on the Panelview.
  MG40:1: This next Message statement is used to send the speed reference to the Powerflex drive.  This speed reference is set by the operator on the Panelview plus.
  C25:1: D E P O S I T     C O U N T
  B23:0/12: Recipe number  x 10 = Recipe data location
    
    example:  Recipe #6 is located in Data location F100:60
    
    Each recipe contains information on
    # of rows
    1st row Distance
    row to row Distance
    Velocity of indexes
  B12:0/13: T O   S I L E N C E   P R E S S   A C K   O R   S I L E N C E   A L A R M   O N   H M I
  U:31: ACCEL REVERSE
  T24:67: M A I N     D E P O S I T
       P V            D E P O S I T
  T24:65: M A I N     S U C T I O N
       P V            D E P O S I T
    
    
      D E P O S I T    S H I F T   D E L A Y
  T24:63: M A I N     S U C T I O N
       P V            S U C T I O N
  T24:60: M E S S A G E    S T A T E M E N T S    T O    B R I D G E    S E R V O    D R I V E
  T24:54: S E R V O   W I L L   A U T O M A T I C A L L Y   H O M E   O N   P O W E R   U P
  T4:21: NC/NF - NO CONTAINER NO FILL LOGIC
    
    THE PAN IS LATCHED IF PRESET AFTER THE FLIGHT IS SEEN BY THE FLIGHT DETECT SENSOR.  HOWEVER THIS LATCH CAN ONLY OCCUR 100ms AFTER THE FLIGHT IS DETECTED.  THIS GIVES THE PLC TIME TO MOVE THE LAST LATCH INTO THE BIT SHIFT.
  T4:20: M E S S A G E    S T A T E M E N T S    T O    B R I D G E    S E R V O    D R I V E
  N97:0: RECIPE BEING MOVED INTO   N 9 0 : ( 0 - 9 )  WITH A ONE SHOT ALLOWS THE OPERATOR TO CHANGE THE EXISTING PARAMETERS WITHOUT CHANGING THE RECIPE PERMANENTLY.

DATA TABLE (non-zero values as saved)
DATA B3
% B3:0 % 0X00BF 0X0005 0X0040 0X0000 0X0000 0X0000 0X0000 0X0000 0X0000 0X0000
DATA T4
% .PRE .ACC %
% T4:0 % 200 0
% T4:1 % 6 0
% T4:2 % 400 0
% T4:3 % 200 0
% T4:4 % 200 0
% T4:5 % 200 200
% T4:6 % 1000 1000
% T4:7 % 5000 0
% T4:8 % 60 60
% T4:9 % 1000 0
% T4:10 % 1000 0
% T4:11 % 300 0
% T4:12 % 300 0
% T4:13 % 300 0
% T4:14 % 300 0
% T4:21 % 10000 0
DATA C5
% .PRE .ACC %
% C5:0 % 4 1
% C5:1 % 10 8
% C5:3 % 99 0
DATA R6
% .LEN .POS %
% R6:0 % 20 0
% R6:1 % 48 0
% R6:2 % 10 9
% R6:3 % 10 9
DATA N7
% N7:0 % 1 131 132 132 133 129 133 131 136 133
% N7:10 % 0 8 0 0 0 0 0 0 0 0
% N7:20 % 0 83 82 81 83 81 82 81 82 82
DATA F8
% F8:0 % 693 550 8 0 0
DATA B11
% B11:0 % 0X5BFB 0X1840 0X0099 0X1C15 0X0154
DATA B12
% B12:0 % 0X44C0 0X0002 0X0000 0X1008 0X0000 0X0000 0X0000 0X0000 0X0000 0X0000
DATA B23
% B23:0 % 0X4801 0X6004 0XBBE0 0X3311 0X21F4 0X2000 0X0000 0X0000 0X0000 0X0000
% B23:10 % 0X0000 0X0000 0X0000 0X0000 0X0000 0X0008 0X0000 0X0000 0X0000 0X0000
DATA T24
% .PRE .ACC %
% T24:0 % 5000 5000
% T24:1 % 500 0
% T24:2 % 2000 0
% T24:3 % 200 0
% T24:4 % 200 200
% T24:5 % 300 0
% T24:6 % 400 52
% T24:7 % 800 52
% T24:8 % 150 150
% T24:9 % 300 220
% T24:10 % 60 52
% T24:11 % 1000 0
% T24:12 % 10000 0
% T24:13 % 2000 0
% T24:14 % 2000 0
% T24:15 % 10000 0
% T24:16 % 10 0
% T24:17 % 10 0
% T24:18 % 10 0
% T24:19 % 2000 0
% T24:20 % 3000 0
% T24:21 % 1000 0
% T24:22 % 1000 0
% T24:23 % 1000 0
% T24:24 % 1000 0
% T24:25 % 1000 0
% T24:26 % 1000 0
% T24:27 % 1000 0
% T24:28 % 1000 0
% T24:29 % 1000 0
% T24:30 % 165 0
% T24:31 % 165 0
% T24:32 % 165 0
% T24:33 % 165 0
% T24:34 % 165 0
% T24:35 % 165 0
% T24:36 % 165 0
% T24:37 % 165 0
% T24:38 % 3000 0
% T24:39 % 500 500
% T24:40 % 165 165
% T24:41 % 165 165
% T24:42 % 165 165
% T24:43 % 165 165
% T24:44 % 165 165
% T24:45 % 165 165
% T24:46 % 165 165
% T24:47 % 165 165
% T24:48 % 10 0
% T24:49 % 3000 0
% T24:50 % 3000 0
% T24:51 % 3000 0
% T24:52 % 100 0
% T24:53 % 200 0
% T24:54 % 10000 0
% T24:55 % 5000 0
% T24:56 % 500 0
% T24:57 % 500 500
% T24:58 % 12000 12000
% T24:60 % 300 0
% T24:65 % 140 0
% T24:69 % 140 0
% T24:72 % 2 0
% T24:82 % 400 400
DATA C25
% .PRE .ACC %
% C25:0 % 1000 0
% C25:1 % 1 0
% C25:2 % 15 0
% C25:3 % 12 1
% C25:5 % 10 0
DATA N27
% N27:0 % 1 2 20 2 1 7 150 150 1 0
% N27:40 % 0 111 222 333 444 555 11112 0 10101 32767
% N27:100 % 0 1 2 3 88 99 99 99 99 99
% N27:110 % 0 99 99 99 99 99 99 99 99 99
% N27:120 % 0 99 99 99 99 99 99 99 99 99
% N27:130 % 0 99 99 99 99 99 99 99 99 99
% N27:140 % 0 99 99 99 99 99 99 99 99 99
% N27:150 % 0 99 99 99 99 99 99 99 99 99
% N27:160 % 0 99 99 99 99 99 99 99 99 99
% N27:170 % 90 99 99 99 99 99 99 99 99 99
DATA F28
% F28:0 % 1 1 1 1 4096
% F28:5 % 25000 0 0 0 0
% F28:10 % 99 250 399 98 0
% F28:20 % 3566 0 0 0 0
